		Funktionstyp:			RHD (kurz für Relative Humidity)
		Instanz-ID:				hier 1 (in XML nachschauen)
		Aktion:					STATUS
		P1:						Relative Luftfeuchtigkeit 0-100 Vorkommastellen
		P2:						Relative Luftfeuchtigkeit 0-100 Nachkommastellen

	Telegram Statusabfrage:  	
	
	\xFD 12345.RHD.1.gSTATUS \xFE
	
	Antwort:  					\xFD 12345.RHD.1.rSTATUS.P1 \xFE
	P1:							Relative Luftfeuchtigkeit 0-100 Vorkommastellen
	P2:							Relative Luftfeuchtigkeit 0-100 Nachkommastellen

	(*------------------------------------------------------------*)
	Helligkeitssensor (Sensor):
	(*------------------------------------------------------------*)
	Telegram Event:  	
	
	\xFD 12345.BRS.23.STATUS.P1.P2 \xFE
	
		Funktionstyp:			BRS (kurz für Brightness Sensor)
		Instanz-ID:				hier 23 (in XML nachschauen)
		Aktion:					STATUS
		P1:						Relative Helligkeit 0-255 Vorkommastellen
		P2:						Relative Helligkeit 0-255 Nachkommastellen
	
	Telegram Statusabfrage:  	
	
	\xFD 12345.BRS.23.gSTATUS \xFE
	
	Antwort:  					\xFD 12345.BRS.23.rSTATUS.P1 \xFE
	P1:							Relative Helligkeit 0-255 Vorkommastellen
	P2:							Relative Helligkeit 0-255 Nachkommastellen

(*======================================================================================================================================*)
(* Alle Telegramme im Überblick *)	

	<?xml version="1.0" encoding="utf-8"?>
	<Comm Title="Haus-Bus ID 1212" Comment="" Baudrate="57600" Databits="8" Parity="1" EndChar="510">
	<CommCmd Title="16-fach Relais 1212 - Rote Modul LED" Comment="" CmdOn="\xFD1212.OUT.210.ON.0\xFE" CmdOff="\xFD1212.OUT.210.OFF\xFE" Unit="" Analog="false" Text="false" Sensor="false" SourceValHigh="100" DestValHigh="100"/>
	<CommCmd Title="16-fach Relais 1212 - Relais 1" Comment="" CmdOn="\xFD1212.OUT.17.ON.0\xFE" CmdOff="\xFD1212.OUT.17.OFF\xFE" Unit="" Analog="false" Text="false" Sensor="false" SourceValHigh="100" DestValHigh="100"/>
	<CommCmd Title="16-fach Relais 1212 - Relais 2" Comment="" CmdOn="\xFD1212.OUT.18.ON.0\xFE" CmdOff="\xFD1212.OUT.18.OFF\xFE" Unit="" Analog="false" Text="false" Sensor="false" SourceValHigh="100" DestValHigh="100"/>
	<CommCmd Title="16-fach Relais 1212 - Relais 3" Comment="" CmdOn="\xFD1212.OUT.19.ON.0\xFE" CmdOff="\xFD1212.OUT.19.OFF\xFE" Unit="" Analog="false" Text="false" Sensor="false" SourceValHigh="100" DestValHigh="100"/>
	<CommCmd Title="16-fach Relais 1212 - Relais 4" Comment="" CmdOn="\xFD1212.OUT.20.ON.0\xFE" CmdOff="\xFD1212.OUT.20.OFF\xFE" Unit="" Analog="false" Text="false" Sensor="false" SourceValHigh="100" DestValHigh="100"/>
	<CommCmd Title="16-fach Relais 1212 - Relais 5" Comment="" CmdOn="\xFD1212.OUT.21.ON.0\xFE" CmdOff="\xFD1212.OUT.21.OFF\xFE" Unit="" Analog="false" Text="false" Sensor="false" SourceValHigh="100" DestValHigh="100"/>
	<CommCmd Title="16-fach Relais 1212 - Relais 6" Comment="" CmdOn="\xFD1212.OUT.22.ON.0\xFE" CmdOff="\xFD1212.OUT.22.OFF\xFE" Unit="" Analog="false" Text="false" Sensor="false" SourceValHigh="100" DestValHigh="100"/>
	<CommCmd Title="16-fach Relais 1212 - Relais 7" Comment="" CmdOn="\xFD1212.OUT.23.ON.0\xFE" CmdOff="\xFD1212.OUT.23.OFF\xFE" Unit="" Analog="false" Text="false" Sensor="false" SourceValHigh="100" DestValHigh="100"/>
	<CommCmd Title="16-fach Relais 1212 - Relais 8" Comment="" CmdOn="\xFD1212.OUT.24.ON.0\xFE" CmdOff="\xFD1212.OUT.24.OFF\xFE" Unit="" Analog="false" Text="false" Sensor="false" SourceValHigh="100" DestValHigh="100"/>
	<CommCmd Title="16-fach Relais 1212 - Relais 9" Comment="" CmdOn="\xFD1212.OUT.33.ON.0\xFE" CmdOff="\xFD1212.OUT.33.OFF\xFE" Unit="" Analog="false" Text="false" Sensor="false" SourceValHigh="100" DestValHigh="100"/>
	<CommCmd Title="16-fach Relais 1212 - Relais 10" Comment="" CmdOn="\xFD1212.OUT.34.ON.0\xFE" CmdOff="\xFD1212.OUT.34.OFF\xFE" Unit="" Analog="false" Text="false" Sensor="false" SourceValHigh="100" DestValHigh="100"/>
	<CommCmd Title="16-fach Relais 1212 - Relais 11" Comment="" CmdOn="\xFD1212.OUT.35.ON.0\xFE" CmdOff="\xFD1212.OUT.35.OFF\xFE" Unit="" Analog="false" Text="false" Sensor="false" SourceValHigh="100" DestValHigh="100"/>
	<CommCmd Title="16-fach Relais 1212 - Relais 12" Comment="" CmdOn="\xFD1212.OUT.36.ON.0\xFE" CmdOff="\xFD1212.OUT.36.OFF\xFE" Unit="" Analog="false" Text="false" Sensor="false" SourceValHigh="100" DestValHigh="100"/>
	<CommCmd Title="16-fach Relais 1212 - Relais 13" Comment="" CmdOn="\xFD1212.OUT.37.ON.0\xFE" CmdOff="\xFD1212.OUT.37.OFF\xFE" Unit="" Analog="false" Text="false" Sensor="false" SourceValHigh="100" DestValHigh="100"/>
	<CommCmd Title="16-fach Relais 1212 - Relais 14" Comment="" CmdOn="\xFD1212.OUT.38.ON.0\xFE" CmdOff="\xFD1212.OUT.38.OFF\xFE" Unit="" Analog="false" Text="false" Sensor="false" SourceValHigh="100" DestValHigh="100"/>
	<CommCmd Title="16-fach Relais 1212 - Relais 15" Comment="" CmdOn="\xFD1212.OUT.39.ON.0\xFE" CmdOff="\xFD1212.OUT.39.OFF\xFE" Unit="" Analog="false" Text="false" Sensor="false" SourceValHigh="100" DestValHigh="100"/>
	<CommCmd Title="16-fach Relais 1212 - Relais 16" Comment="" CmdOn="\xFD1212.OUT.40.ON.0\xFE" CmdOff="\xFD1212.OUT.40.OFF\xFE" Unit="" Analog="false" Text="false" Sensor="false" SourceValHigh="100" DestValHigh="100"/>
	<CommCmd Title="16-fach Relais 1212 - Eingang 1" Comment="" CmdOn="\xFD1212.BTN.97.STATUS.\v\xFE" CmdOff="" Unit="&lt;v.x&gt;" Analog="true" Text="false" Sensor="true" SourceValHigh="100" DestValHigh="100"/>
	<CommCmd Title="16-fach Relais 1212 - Eingang 2" Comment="" CmdOn="\xFD1212.BTN.98.STATUS.\v\xFE" CmdOff="" Unit="&lt;v.x&gt;" Analog="true" Text="false" Sensor="true" SourceValHigh="100" DestValHigh="100"/>
	<CommCmd Title="16-fach Relais 1212 - Eingang 3" Comment="" CmdOn="\xFD1212.BTN.99.STATUS.\v\xFE" CmdOff="" Unit="&lt;v.x&gt;" Analog="true" Text="false" Sensor="true" SourceValHigh="100" DestValHigh="100"/>
	<CommCmd Title="16-fach Relais 1212 - Eingang 4" Comment="" CmdOn="\xFD1212.BTN.100.STATUS.\v\xFE" CmdOff="" Unit="&lt;v.x&gt;" Analog="true" Text="false" Sensor="true" SourceValHigh="100" DestValHigh="100"/>
	<CommCmd Title="16-fach Relais 1212 - Eingang 5" Comment="" CmdOn="\xFD1212.BTN.101.STATUS.\v\xFE" CmdOff="" Unit="&lt;v.x&gt;" Analog="true" Text="false" Sensor="true" SourceValHigh="100" DestValHigh="100"/>
	<CommCmd Title="16-fach Relais 1212 - Eingang 6" Comment="" CmdOn="\xFD1212.BTN.102.STATUS.\v\xFE" CmdOff="" Unit="&lt;v.x&gt;" Analog="true" Text="false" Sensor="true" SourceValHigh="100" DestValHigh="100"/>
	<CommCmd Title="16-fach Relais 1212 - Eingang 7" Comment="" CmdOn="\xFD1212.BTN.103.STATUS.\v\xFE" CmdOff="" Unit="&lt;v.x&gt;" Analog="true" Text="false" Sensor="true" SourceValHigh="100" DestValHigh="100"/>
	<CommCmd Title="16-fach Relais 1212 - Eingang 8" Comment="" CmdOn="\xFD1212.BTN.104.STATUS.\v\xFE" CmdOff="" Unit="&lt;v.x&gt;" Analog="true" Text="false" Sensor="true" SourceValHigh="100" DestValHigh="100"/>
	</Comm>

*)
END_ACTION

END_FUNCTION_BLOCK

// ---- POUs/RS485_Hausbus_FB/RelaisModul/fb_StringConvRB16F.TcPOU
(*======================================================================================================================================*)
(*fb_StringConvRB16F:	Zusammensetzen des Strings für 16Fach Bus Relaismodul		*)
(*
Date          	| Version    	| created under        	| Author          	| Remark *)
(*====================================================================================================================================================*)
(*08/05/2025   	| 1.00      		| TC3		  		| N.Kersting       | first release *)
(*====================================================================================================================================================*)
FUNCTION_BLOCK fb_StringConvRB16F
VAR_INPUT
	I_bReset			:BOOL;							(* Reset Befehl auslösen *)
	I_bRedLEDOn			:BOOL;							(* Schaltet nur die Rote Modul LED ein*)
	I_bRedLEDOff		:BOOL;							(* Schaltet nur die Rote Modul LED aus*)
	I_diID				:DINT;							(* Device ID *)
	I_bOut    	 		:ARRAY[1..16] OF BOOL;     	  	(* gewünschter Relais zustand (TRUE = An %)*)
	
	I_iSection			:INT :=1;							(* Paarweise Schalten 1= 1&2 2= 3&4 usw. *)
	
	I_sStartZeichen		:BYTE := 16#FD;					(* Startzeichen Präfix *)
	I_sEndZeichen		:BYTE := 16#FE;					(* Endzeichen Suffix *)
END_VAR
VAR_OUTPUT
	Q_sConvString		:STRING(255);
END_VAR
VAR
	iStartOut			:INT := 1;
	iStartInstIDExt		:INT :=65;
	
END_VAR

IF NOT I_bReset
THEN
	IF I_bRedLEDOn
	THEN
		(* Rote Modul LED Ein*)
		iStartInstIDExt := 210;
		
		Q_sConvString:=	CONCAT(F_ToCHR(I_sStartZeichen),DINT_TO_STRING(I_diID));
		Q_sConvString:=	CONCAT(Q_sConvString,'.OUT.');
		Q_sConvString:=	CONCAT(Q_sConvString,INT_TO_STRING(iStartInstIDExt));
		Q_sConvString:=	CONCAT(Q_sConvString,'.ON');
		Q_sConvString:=	CONCAT(Q_sConvString,F_ToCHR(I_sEndZeichen));
	ELSIF
		I_bRedLEDOff
	THEN
		(* Rote Modul LED Aus*)
		iStartInstIDExt := 210;
		
		Q_sConvString:=	CONCAT(F_ToCHR(I_sStartZeichen),DINT_TO_STRING(I_diID));
		Q_sConvString:=	CONCAT(Q_sConvString,'.OUT.');
		Q_sConvString:=	CONCAT(Q_sConvString,INT_TO_STRING(iStartInstIDExt));
		Q_sConvString:=	CONCAT(Q_sConvString,'.OFF');
		Q_sConvString:=	CONCAT(Q_sConvString,F_ToCHR(I_sEndZeichen));
	ELSE
		CASE I_iSection OF
			
		0:	Q_sConvString:='';
		
		1:	(* 1 & 2 Schalten *)
			iStartInstIDExt := 17;
			iStartOut :=	1;
			
			Q_sConvString:=	CONCAT(F_ToCHR(I_sStartZeichen),DINT_TO_STRING(I_diID));
			Q_sConvString:=	CONCAT(Q_sConvString,'.OUT.');
			Q_sConvString:=	CONCAT(Q_sConvString,INT_TO_STRING(iStartInstIDExt));
			IF I_bOut[iStartOut]
			THEN
				Q_sConvString:=	CONCAT(Q_sConvString,'.ON');
			ELSE
				Q_sConvString:=	CONCAT(Q_sConvString,'.OFF');
			END_IF
			Q_sConvString:=	CONCAT(Q_sConvString,F_ToCHR(I_sEndZeichen));
			
			(* ##2 ##*)
			iStartInstIDExt := iStartInstIDExt +1;
			iStartOut:= iStartOut+1;
			
			Q_sConvString:=	CONCAT(Q_sConvString,F_ToCHR(I_sStartZeichen));
			Q_sConvString:=	CONCAT(Q_sConvString,DINT_TO_STRING(I_diID));
			Q_sConvString:=	CONCAT(Q_sConvString,'.OUT.');
			Q_sConvString:=	CONCAT(Q_sConvString,INT_TO_STRING(iStartInstIDExt));
			IF I_bOut[iStartOut]
			THEN
				Q_sConvString:=	CONCAT(Q_sConvString,'.ON');
			ELSE
				Q_sConvString:=	CONCAT(Q_sConvString,'.OFF');
			END_IF
			Q_sConvString:=	CONCAT(Q_sConvString,F_ToCHR(I_sEndZeichen));
		
			(* ##3 ##*)
			iStartInstIDExt := iStartInstIDExt +1;
			iStartOut:= iStartOut+1;
			
			Q_sConvString:=	CONCAT(Q_sConvString,F_ToCHR(I_sStartZeichen));
			Q_sConvString:=	CONCAT(Q_sConvString,DINT_TO_STRING(I_diID));
			Q_sConvString:=	CONCAT(Q_sConvString,'.OUT.');
			Q_sConvString:=	CONCAT(Q_sConvString,INT_TO_STRING(iStartInstIDExt));
			IF I_bOut[iStartOut]
			THEN
				Q_sConvString:=	CONCAT(Q_sConvString,'.ON');
			ELSE
				Q_sConvString:=	CONCAT(Q_sConvString,'.OFF');
			END_IF
			Q_sConvString:=	CONCAT(Q_sConvString,F_ToCHR(I_sEndZeichen));
			
			(* ##4 ##*)
			iStartInstIDExt := iStartInstIDExt +1;
			iStartOut:= iStartOut+1;
			
			Q_sConvString:=	CONCAT(Q_sConvString,F_ToCHR(I_sStartZeichen));
			Q_sConvString:=	CONCAT(Q_sConvString,DINT_TO_STRING(I_diID));
			Q_sConvString:=	CONCAT(Q_sConvString,'.OUT.');
			Q_sConvString:=	CONCAT(Q_sConvString,INT_TO_STRING(iStartInstIDExt));
			IF I_bOut[iStartOut]
			THEN
				Q_sConvString:=	CONCAT(Q_sConvString,'.ON');
			ELSE
				Q_sConvString:=	CONCAT(Q_sConvString,'.OFF');
			END_IF
			Q_sConvString:=	CONCAT(Q_sConvString,F_ToCHR(I_sEndZeichen));
		
			(* ##5 ##*)
			iStartInstIDExt := iStartInstIDExt +1;
			iStartOut:= iStartOut+1;
			
			Q_sConvString:=	CONCAT(Q_sConvString,F_ToCHR(I_sStartZeichen));
			Q_sConvString:=	CONCAT(Q_sConvString,DINT_TO_STRING(I_diID));
			Q_sConvString:=	CONCAT(Q_sConvString,'.OUT.');
			Q_sConvString:=	CONCAT(Q_sConvString,INT_TO_STRING(iStartInstIDExt));
			IF I_bOut[iStartOut]
			THEN
				Q_sConvString:=	CONCAT(Q_sConvString,'.ON');
			ELSE
				Q_sConvString:=	CONCAT(Q_sConvString,'.OFF');
			END_IF
			Q_sConvString:=	CONCAT(Q_sConvString,F_ToCHR(I_sEndZeichen));
			
			(* ##6 ##*)
			iStartInstIDExt := iStartInstIDExt +1;
			iStartOut:= iStartOut+1;
			
			Q_sConvString:=	CONCAT(Q_sConvString,F_ToCHR(I_sStartZeichen));
			Q_sConvString:=	CONCAT(Q_sConvString,DINT_TO_STRING(I_diID));
			Q_sConvString:=	CONCAT(Q_sConvString,'.OUT.');
			Q_sConvString:=	CONCAT(Q_sConvString,INT_TO_STRING(iStartInstIDExt));
			IF I_bOut[iStartOut]
			THEN
				Q_sConvString:=	CONCAT(Q_sConvString,'.ON');
			ELSE
				Q_sConvString:=	CONCAT(Q_sConvString,'.OFF');
			END_IF
			Q_sConvString:=	CONCAT(Q_sConvString,F_ToCHR(I_sEndZeichen));
		
			(* ##7 ##*)
			iStartInstIDExt := iStartInstIDExt +1;
			iStartOut:= iStartOut+1;
			
			Q_sConvString:=	CONCAT(Q_sConvString,F_ToCHR(I_sStartZeichen));
			Q_sConvString:=	CONCAT(Q_sConvString,DINT_TO_STRING(I_diID));
			Q_sConvString:=	CONCAT(Q_sConvString,'.OUT.');
			Q_sConvString:=	CONCAT(Q_sConvString,INT_TO_STRING(iStartInstIDExt));
			IF I_bOut[iStartOut]
			THEN
				Q_sConvString:=	CONCAT(Q_sConvString,'.ON');
			ELSE
				Q_sConvString:=	CONCAT(Q_sConvString,'.OFF');
			END_IF
			Q_sConvString:=	CONCAT(Q_sConvString,F_ToCHR(I_sEndZeichen));
			
			(* ##8 ##*)
			iStartInstIDExt := iStartInstIDExt +1;
			iStartOut:= iStartOut+1;
			
			Q_sConvString:=	CONCAT(Q_sConvString,F_ToCHR(I_sStartZeichen));
			Q_sConvString:=	CONCAT(Q_sConvString,DINT_TO_STRING(I_diID));
			Q_sConvString:=	CONCAT(Q_sConvString,'.OUT.');
			Q_sConvString:=	CONCAT(Q_sConvString,INT_TO_STRING(iStartInstIDExt));
			IF I_bOut[iStartOut]
			THEN
				Q_sConvString:=	CONCAT(Q_sConvString,'.ON');
			ELSE
				Q_sConvString:=	CONCAT(Q_sConvString,'.OFF');
			END_IF
			Q_sConvString:=	CONCAT(Q_sConvString,F_ToCHR(I_sEndZeichen));
		
		2:	(* 9 & 10 Schalten *)
			iStartInstIDExt := 33;
			iStartOut :=	9;
			
			Q_sConvString:=	CONCAT(F_ToCHR(I_sStartZeichen),DINT_TO_STRING(I_diID));
			Q_sConvString:=	CONCAT(Q_sConvString,'.OUT.');
			Q_sConvString:=	CONCAT(Q_sConvString,INT_TO_STRING(iStartInstIDExt));
			IF I_bOut[iStartOut]
			THEN
				Q_sConvString:=	CONCAT(Q_sConvString,'.ON');
			ELSE
				Q_sConvString:=	CONCAT(Q_sConvString,'.OFF');
			END_IF
			Q_sConvString:=	CONCAT(Q_sConvString,F_ToCHR(I_sEndZeichen));
			
			(* ##10 ##*)
			iStartInstIDExt := iStartInstIDExt +1;
			iStartOut:= iStartOut+1;
			
			Q_sConvString:=	CONCAT(Q_sConvString,F_ToCHR(I_sStartZeichen));
			Q_sConvString:=	CONCAT(Q_sConvString,DINT_TO_STRING(I_diID));
			Q_sConvString:=	CONCAT(Q_sConvString,'.OUT.');
			Q_sConvString:=	CONCAT(Q_sConvString,INT_TO_STRING(iStartInstIDExt));
			IF I_bOut[iStartOut]
			THEN
				Q_sConvString:=	CONCAT(Q_sConvString,'.ON');
			ELSE
				Q_sConvString:=	CONCAT(Q_sConvString,'.OFF');
			END_IF
			Q_sConvString:=	CONCAT(Q_sConvString,F_ToCHR(I_sEndZeichen));
		
			(* ##11 ##*)
			iStartInstIDExt := iStartInstIDExt +1;
			iStartOut:= iStartOut+1;
			
			Q_sConvString:=	CONCAT(Q_sConvString,F_ToCHR(I_sStartZeichen));
			Q_sConvString:=	CONCAT(Q_sConvString,DINT_TO_STRING(I_diID));
			Q_sConvString:=	CONCAT(Q_sConvString,'.OUT.');
			Q_sConvString:=	CONCAT(Q_sConvString,INT_TO_STRING(iStartInstIDExt));
			IF I_bOut[iStartOut]
			THEN
				Q_sConvString:=	CONCAT(Q_sConvString,'.ON');
			ELSE
				Q_sConvString:=	CONCAT(Q_sConvString,'.OFF');
			END_IF
			Q_sConvString:=	CONCAT(Q_sConvString,F_ToCHR(I_sEndZeichen));
			
			(* ##12 ##*)
			iStartInstIDExt := iStartInstIDExt +1;
			iStartOut:= iStartOut+1;
			
			Q_sConvString:=	CONCAT(Q_sConvString,F_ToCHR(I_sStartZeichen));
			Q_sConvString:=	CONCAT(Q_sConvString,DINT_TO_STRING(I_diID));
			Q_sConvString:=	CONCAT(Q_sConvString,'.OUT.');
			Q_sConvString:=	CONCAT(Q_sConvString,INT_TO_STRING(iStartInstIDExt));
			IF I_bOut[iStartOut]
			THEN
				Q_sConvString:=	CONCAT(Q_sConvString,'.ON');
			ELSE
				Q_sConvString:=	CONCAT(Q_sConvString,'.OFF');
			END_IF
			Q_sConvString:=	CONCAT(Q_sConvString,F_ToCHR(I_sEndZeichen));
		
			(* ##13 ##*)
			iStartInstIDExt := iStartInstIDExt +1;
			iStartOut:= iStartOut+1;
			
			Q_sConvString:=	CONCAT(Q_sConvString,F_ToCHR(I_sStartZeichen));
			Q_sConvString:=	CONCAT(Q_sConvString,DINT_TO_STRING(I_diID));
			Q_sConvString:=	CONCAT(Q_sConvString,'.OUT.');
			Q_sConvString:=	CONCAT(Q_sConvString,INT_TO_STRING(iStartInstIDExt));
			IF I_bOut[iStartOut]
			THEN
				Q_sConvString:=	CONCAT(Q_sConvString,'.ON');
			ELSE
				Q_sConvString:=	CONCAT(Q_sConvString,'.OFF');
			END_IF
			Q_sConvString:=	CONCAT(Q_sConvString,F_ToCHR(I_sEndZeichen));
			
			(* ##14 ##*)
			iStartInstIDExt := iStartInstIDExt +1;
			iStartOut:= iStartOut+1;
			
			Q_sConvString:=	CONCAT(Q_sConvString,F_ToCHR(I_sStartZeichen));
			Q_sConvString:=	CONCAT(Q_sConvString,DINT_TO_STRING(I_diID));
			Q_sConvString:=	CONCAT(Q_sConvString,'.OUT.');
			Q_sConvString:=	CONCAT(Q_sConvString,INT_TO_STRING(iStartInstIDExt));
			IF I_bOut[iStartOut]
			THEN
				Q_sConvString:=	CONCAT(Q_sConvString,'.ON');
			ELSE
				Q_sConvString:=	CONCAT(Q_sConvString,'.OFF');
			END_IF
			Q_sConvString:=	CONCAT(Q_sConvString,F_ToCHR(I_sEndZeichen));
		
			(* ##15 ##*)
			iStartInstIDExt := iStartInstIDExt +1;
			iStartOut:= iStartOut+1;
			
			Q_sConvString:=	CONCAT(Q_sConvString,F_ToCHR(I_sStartZeichen));
			Q_sConvString:=	CONCAT(Q_sConvString,DINT_TO_STRING(I_diID));
			Q_sConvString:=	CONCAT(Q_sConvString,'.OUT.');
			Q_sConvString:=	CONCAT(Q_sConvString,INT_TO_STRING(iStartInstIDExt));
			IF I_bOut[iStartOut]
			THEN
				Q_sConvString:=	CONCAT(Q_sConvString,'.ON');
			ELSE
				Q_sConvString:=	CONCAT(Q_sConvString,'.OFF');
			END_IF
			Q_sConvString:=	CONCAT(Q_sConvString,F_ToCHR(I_sEndZeichen));
			
			(* ##16 ##*)
			iStartInstIDExt := iStartInstIDExt +1;
			iStartOut:= iStartOut+1;
			
			Q_sConvString:=	CONCAT(Q_sConvString,F_ToCHR(I_sStartZeichen));
			Q_sConvString:=	CONCAT(Q_sConvString,DINT_TO_STRING(I_diID));
			Q_sConvString:=	CONCAT(Q_sConvString,'.OUT.');
			Q_sConvString:=	CONCAT(Q_sConvString,INT_TO_STRING(iStartInstIDExt));
			IF I_bOut[iStartOut]
			THEN
				Q_sConvString:=	CONCAT(Q_sConvString,'.ON');
			ELSE
				Q_sConvString:=	CONCAT(Q_sConvString,'.OFF');
			END_IF
			Q_sConvString:=	CONCAT(Q_sConvString,F_ToCHR(I_sEndZeichen));
		END_CASE
	END_IF
	
ELSE
	(* Reset *)
	Q_sConvString:=	CONCAT(F_ToCHR(I_sStartZeichen),DINT_TO_STRING(I_diID));
	Q_sConvString:=	CONCAT(Q_sConvString,'.SYS.');
	Q_sConvString:=	CONCAT(Q_sConvString,INT_TO_STRING(1));
	Q_sConvString:=	CONCAT(Q_sConvString,'.RESET');
	Q_sConvString:=	CONCAT(Q_sConvString,F_ToCHR(I_sEndZeichen));
END_IF

END_FUNCTION_BLOCK

// ---- POUs/RS485_Hausbus_FB/RS485 COM/RS485_Master/fb_RS485Startup.TcPOU
(*======================================================================================================================================*)
(*fb_RS485Startup:	Einfacher Baustein um die Hardware für die RS485 Haus-Bus vorzubereiten*)
(*
Date          	| Version    	| created under        	| Author          	| Remark *)
(*====================================================================================================================================================*)
(*13/05/2025   	| 1.00      		| TC3		  		| N.Kersting       | first release *)
(*====================================================================================================================================================*)
FUNCTION_BLOCK fb_RS485Startup
VAR_INPUT
	I_bExecute						:BOOL;
	I_bBusOK						:BOOL;
	I_tStartupVerz					:TIME := T#2S;	(* Startup verzögert ausführen *)
END_VAR
VAR_IN_OUT
	IQ_InData	 					:KL6inData22B;
    IQ_OutData						:KL6outData22B;
END_VAR
VAR_OUTPUT
	Q_sState						:STRING;
	Q_bStartupDone					:BOOL;
	Q_bError						:BOOL;
	Q_stStates						:ST_RS485Startup_State;
END_VAR
VAR
	udBaudrate						:UDINT := 57600;
	byDataBits						:BYTE := 8;
	byStopBits						:BYTE := 1;
	
	tonStartupVerz					:ton;
	fbSerialComReset				:ComReset;
	fComBufferReset					:ClearComBuffer;
	fbSerialConfig 					:KL6Configuration;  // Terminal-Konfiguration (Baud, Parität etc.)
	iStepStartup					:INT;
END_VAR

tonStartupVerz(
	PT :=	I_tStartupVerz);
	
CASE iStepStartup OF 
(*=========================================================================*)
0:	IF NOT Q_bError
		AND I_bBusOK
	THEN
		Q_sState := 'INIT';
	ELSIF
		NOT I_bBusOK
	THEN
		Q_bError := TRUE;
		Q_sState := 'Busverbindung nicht Ok';
	END_IF
	
	tonStartupVerz.IN := FALSE;
	
	fbSerialComReset(
		Execute:= 		FALSE);
		
	fbSerialConfig(
		Execute:= 		FALSE);
		
	IF I_bExecute
		AND I_bBusOK
	THEN
		Q_bStartupDone := FALSE;
		iStepStartup := iStepStartup+1;
	END_IF

(*=========================================================================*)
1:	Q_sState := 'Warten auf Verzögerung';
	tonStartupVerz.IN := TRUE; 
	
	IF tonStartupVerz.Q
	THEN
		iStepStartup := iStepStartup+1;
	END_IF
	
(*=========================================================================*)
2:	Q_sState := 'Serielle Klemme Konfigurieren mit Haus-Bus Vorgaben';	
	
	fbSerialConfig(
		Execute:= 		TRUE, 
		Mode:= 			ComSerialLineMode_t.SERIALLINEMODE_KL6_22B_STANDARD,		 
		Baudrate:= 		udBaudrate, 
		NoDatabits:= 	byDataBits, 
		Parity:= 		ComParity_t.PARITY_EVEN,	 
		Stopbits:= 		byStopBits, 
		Handshake:= 	RS485_HALFDUPLEX, 
		ContinousMode:= , 
		pComIn := 		ADR(IQ_InData), 
		pComOut := 		ADR(IQ_OutData), 
		SizeComIn := 	SIZEOF(IQ_InData),
		Done=> , 
		Busy=> , 
		Error=> , 
		ErrorId=> );
	
	IF fbSerialConfig.Done
	THEN
		fbSerialConfig(
			Execute:= 		FALSE); 
			
		iStepStartup := 3;
	ELSIF
		fbSerialConfig.Error
	THEN
		Q_sState := 'Error fbSerialConfig ID: ';
		Q_sState := CONCAT(Q_sState,INT_TO_STRING(fbSerialConfig.ErrorID));
		iStepStartup := -2;	//Error
	END_IF

(*=========================================================================*)
3:	Q_sState := 'Serielle Klemme Reset Auführen';	
		
	fbSerialComReset(
		Execute:= 		TRUE, 
		pComIn := 		ADR(IQ_InData), 
		pComOut := 		ADR(IQ_OutData), 
		SizeComIn := 	SIZEOF(IQ_InData),
		Done=> , 
		Busy=> , 
		Error=> , 
		ErrorID=> );	
		
	IF fbSerialComReset.Done
	THEN
		iStepStartup := 999;
	ELSIF
		fbSerialComReset.Error
	THEN
		Q_sState := 'Error fbSerialComReset ID: ';
		Q_sState := CONCAT(Q_sState,INT_TO_STRING(fbSerialComReset.ErrorID));
		iStepStartup := -3;	//Error
	END_IF
	
(*=========================================================================*)
999:Q_sState := 'Startup Ausgeführt!';	
	Q_bStartupDone := TRUE;
	Q_bError := FALSE;
	
	IF NOT I_bBusOK
	THEN
		Q_bStartupDone := FALSE;
		iStepStartup := 0;
	END_IF

ELSE
	(* ERROR *)
	Q_bError := TRUE;
	iStepStartup := 0;
END_CASE

(* StatusStruktur für Visu *)
Q_stStates.bBusOk				:=	I_bBusOK;
Q_stStates.bStartupDone			:=	Q_bStartupDone;
Q_stStates.bStartupError		:=	Q_bError;
Q_stStates.sStartupState		:=	Q_sState;

END_FUNCTION_BLOCK

// ---- POUs/RS485_Hausbus_FB/RS485 COM/RS485_Master/fb_RS485FiFoMaster.TcPOU
(*======================================================================================================================================*)
(*fb_RS485FiFoMaster:	Einfaches Senden eines Telegrams über RS485*)
(*
Date          	| Version    	| created under        	| Author          	| Remark *)
(*====================================================================================================================================================*)
(*10/05/2025   	| 1.00      		| TC3		  		| N.Kersting       | first release *)
(*10/05/2025   	| 1.01      		| TC3		  		| N.Kersting       | Nun wird der Empfang auch mit Implementiert  *)
(*13/05/2025   	| 1.02      		| TC3		  		| N.Kersting       | Busbelastungstest Implementiert - Sendet Durchgehend Strings *)
(*14/05/2025   	| 1.03      		| TC3		  		| N.Kersting       | Busauslastung direkt Implementiert *)
(*====================================================================================================================================================*)
FUNCTION_BLOCK fb_RS485FiFoMaster
VAR_INPUT
	I_sSendCmdFiFo				:ARRAY[1..cMaxRS485CMDFiFo] OF STRING(255);
	I_bExecute					:BOOL := TRUE;
	I_bBusBelastungstest		:BOOL;
	I_bReset					:BOOL;
	I_pTxBuffer					:POINTER TO ComBuffer;  (*Zeiger auf TX-Buffer*)
	I_pRxBuffer   				:POINTER TO ComBuffer;  (*Zeiger auf RX-Buffer*)
END_VAR
VAR_OUTPUT
	Q_sReceiveString			:STRING(255);		
	Q_lrBusAuslastung			:LREAL;
	Q_bBusy						:BOOL;
	Q_bDone						:BOOL;
	Q_bError					:BOOL;
	Q_sState					:STRING;
	Q_stStates					:ST_FiFoMaster_State;
END_VAR
VAR
	bFirstCycle					:BOOL := TRUE;
	tVerzReceive				:TIME := T#30MS;			(* Zeit, die zum Empfangen bleibt *)
	
	tonSend						:ton;
	fbSend     					:SendString255;
	fbReceive   				:ReceiveString255;
	sStartZeichen				:BYTE := 16#FD;				(* Startzeichen Präfix *)
	sEndZeichen					:BYTE := 16#FE;				(* Endzeichen Suffix *)
	sReceivedMEMString			:STRING(255);
	sReceivedString				:STRING(255);
	iStep						:INT;
	iStepReceive				:INT;
	iMaxBufferBlocking			:INT := 0;
	bBusyMem					:BOOL;
	sStep						:STRING;
	sString						:STRING(255);
	sStringSend					:STRING(255);
	tonVerzReceive				:ton;	
	tonTimeout					:ton;
	bStringSend					:BOOL := FALSE;
	icntError					:INT;
	
	iFiFoRow					:INT := 1;
	icntFiFo					:INT;
	i,h							:INT;
	iStepFiFo					:INT;
	
	bBusBelastungstest			:BOOL := FALSE;
	bBusAuslastung				:BOOL := TRUE;
	fbBusAuslastung				:fb_FilterArray;
END_VAR

(*============================================================================================*)
tonTimeout(
	PT:=T#1S);
	
tonVerzReceive(
	pt := tVerzReceive);

(* Busbelastungstest *)	
bBusBelastungstest := I_bBusBelastungstest;

sReceivedMEMString:='';
(*============================================================================================*)	
icntFiFo := 0;
FOR i := 1 TO cMaxRS485CMDFiFo BY 1 DO 
	IF (I_sSendCmdFiFo[i]<> '')
	THEN
		icntFiFo := icntFiFo +1;
	END_IF
END_FOR

(*============================================================================================*)
CASE iStepFiFo OF
-1:	sStep := 'FiFo INIT';
	bFirstCycle := FALSE;
	Q_bBusy := FALSE;
	iFiFoRow := 1;
	
	FOR h := 1 TO cMaxRS485CMDFiFo BY 1 DO
		GVL_RS485FiFoSend.bSendDoneFiFo[h] :=TRUE;
	END_FOR
	
	iStepFiFo := 0;

(*============================================================================================*)
0:	sStep := 'Warten, dass FiFo gefüllt wird';
	iFiFoRow := 1;
	bStringSend := FALSE;
	Q_bBusy := FALSE;
	tonVerzReceive.IN := (I_pTxBuffer^.Count<= INT_TO_UINT(iMaxBufferBlocking));
	
	IF (icntFiFo > 0
		OR  bBusBelastungstest)
		AND NOT bFirstCycle
		AND NOT fbReceive.StringReceived
		AND tonVerzReceive.Q
	THEN
		Q_bBusy := TRUE;
		iStepFiFo := 1;
	ELSIF
		bFirstCycle
	THEN
		iStepFiFo := -1;
	END_IF
	
(*============================================================================================*)	
1:	sStep := 'Prüfen ob STRING in FiFo Zeile gefüllt*';
	sStringSend :=	I_sSendCmdFiFo[iFiFoRow]; 
	
	(* Prüfen ob in der ausgewählten Zeile etwas steht *)
	IF I_sSendCmdFiFo[iFiFoRow] = ''
	THEN
		IF iFiFoRow < cMaxRS485CMDFiFo
		THEN
			iFiFoRow := iFiFoRow+1; (* Nächste Zeile, bis etwas drin Steht *)
		ELSE
			IF bBusBelastungstest
			THEN
				sStringSend :=	CONCAT(F_ToCHR(sStartZeichen),'ServiceTOOL-BUSBELASTUNGSTEST-BURSTFIREMODE');
				sStringSend :=	CONCAT(sStringSend,F_ToCHR(sEndZeichen));
				(* Senden *)
				
				IF NOT I_pTxBuffer^.blocked
					AND (I_pTxBuffer^.Error=0)
					AND NOT fbReceive.StringReceived
				THEN
					sStep := 'Prüfe ob Senden noch aktiv ist';
					bStringSend := TRUE;
					sString :=	sStringSend;
					Q_bDone := FALSE;
					Q_bError := FALSE;
					iStepFiFo := iStepFiFo+1;
				END_IF
			ELSE
				iStepFiFo := 0;	(* Alle Zeilen Abgearbeitet *)
			END_IF
			
		END_IF
	ELSE
		(* Senden *)
		GVL_RS485FiFoSend.bSendDoneFiFo[iFiFoRow] :=FALSE;
		
		IF NOT I_pTxBuffer^.blocked
			AND (I_pTxBuffer^.Error=0)
			AND NOT fbReceive.StringReceived
		THEN
			sStep := 'Prüfe ob Senden noch aktiv ist';
			bStringSend := TRUE;
			sString :=	sStringSend;
			Q_bDone := FALSE;
			Q_bError := FALSE;
			iStepFiFo := iStepFiFo+1;
		END_IF
	END_IF
	
(*============================================================================================*)		
2:	sStep := 'Starte Senden';
	Q_bBusy := TRUE;
	tonTimeout.IN := fbSend.Busy;
	
	IF NOT fbSend.Busy
		AND NOT fbReceive.StringReceived
	THEN
		tonSend.IN := FALSE;
		bStringSend := FALSE;
		iStepFiFo := iStepFiFo+1;
	ELSIF
		(fbSend.Error >0)
		AND NOT (fbSend.Error = 2)
	THEN
		sStep := CONCAT('ERROR-',sStep);
		sStep := CONCAT(sStep,'- ');
		sStep := CONCAT(sStep,INT_TO_STRING(fbSend.Error));
		iStepFiFo := -2;
	ELSIF
		tonTimeout.Q
	THEN
		sStep := CONCAT('ERROR- Timeout',sStep);
		iStepFiFo := -2;
	END_IF

3:	(* Senden*)		
	GVL_RS485FiFoSend.bSendDoneFiFo[iFiFoRow] :=TRUE;
	
	IF iFiFoRow < iFiFoRow
	THEN
		iFiFoRow := iFiFoRow+1;
		iStepFiFo := 1;
	ELSE
		Q_bDone := TRUE;
		iStepFiFo := 0;
	END_IF

ELSE
(*============================================================================================*)
	Q_bError := TRUE;
	Q_bBusy := FALSE;
	bBusyMem := FALSE;
	tonTimeout.IN := FALSE;
	
	IF I_bReset
	THEN
		iStepFiFo := 0;
	END_IF
END_CASE

IF bStringSend
THEN
	fbSend(
		SendString:= 	sString,
		TXbuffer:= 		I_pTxBuffer^);
ELSE
	(* Empfangen *)
	ac00_Receive();
END_IF

(* Empfangsmerker 0 Setzen am ende Eines Zyklus *)
Q_sReceiveString := sReceivedMEMString;

(* Busauslastung tracken*)
ac99_Diagnose();

Q_sState :=	sStep;

(* StatusStruktur für Visu *)
Q_stStates.bBusy				:=	Q_bBusy;
Q_stStates.bDone				:=	Q_bDone;
Q_stStates.bError				:=	Q_bError;
Q_stStates.iFiFoCount			:=	icntFiFo;
Q_stStates.iFiFoRow				:=	iFiFoRow;
Q_stStates.lrBusAuslastung		:=	Q_lrBusAuslastung;
Q_stStates.sReceiveString 		:=	Q_sReceiveString;
Q_stStates.sSendString 			:=	sString;
Q_stStates.sState 				:=	Q_sState;

ACTION ac00_Receive:
(* Empfangen *)
CASE iStepReceive OF		
0:	fbReceive(
		Prefix := 			F_ToCHR(sStartZeichen),
		Suffix := 			F_ToCHR(sEndZeichen),
		Timeout:= , 
		Reset:= , 
		StringReceived=> , 
		Busy=> , 
		Error=> , 
		RxTimeout=> , 
		ReceivedString:= 	sReceivedString, 
		RXbuffer:= 			I_pRxBuffer^);
		
	IF fbReceive.StringReceived
	THEN
		iStepReceive := 1;
		sReceivedMEMString := sReceivedString;
	END_IF
	
1:	sReceivedString := '';
	iStepReceive := 0;
	
END_CASE
END_ACTION

ACTION ac99_Diagnose:
(* Busauslastung Prüfen *)
fbBusAuslastung(
	I_bExcecute:= 	bBusAuslastung, 
	I_nWert:= 		UINT_TO_LREAL(I_pTxBuffer^.Count), 
	I_nFilterWert:= 50, 
	Q_nFilter=> 	Q_lrBusAuslastung);
END_ACTION

END_FUNCTION_BLOCK

// ---- POUs/RS485_Hausbus_FB/RS485 COM/FB/fb_FilterArray.TcPOU
(*======================================================================================================================================*)
(* Dieser Baustein Filtert eine Lreal Variable durch bildung eines Mittelwerts
(*======================================================================================================================================*)						

Date          		| Version    		| created under        		| Author          		| Remark *)
(*======================================================================================================================================*)
(*´10/07/2024   	| 1.00      			| TC2			  		| N.Kersting       	| first release *)
(*´15/07/2024   	| 1.01      			| TC2			  		| N.Kersting       	| Filterung nun Variabel einstellbar *)
(*======================================================================================================================================*)
FUNCTION_BLOCK fb_FilterArray
VAR_INPUT
	I_bExcecute	:BOOL;
	I_nWert		:LREAL;
	I_nFilterWert	:INT	:= 10;
END_VAR
VAR_OUTPUT
	Q_nFilter		:LREAL;
END_VAR
VAR
	i	:INT;
	nWertArray	:ARRAY [0..50] OF LREAL;
END_VAR

IF I_bExcecute THEN
   (* // Verschieben der Werte im Array*)
    FOR i := I_nFilterWert - 1 TO 1 BY -1 DO
        nWertArray[i] := nWertArray[i - 1];
    END_FOR

   (* // Neuen Wert einfügen	*)
    nWertArray[0] := I_nWert;

  (*  // Berechnung des gefilterten Wertes*)
    Q_nFilter := 0;
    FOR i := 0 TO I_nFilterWert - 1 DO
        Q_nFilter := Q_nFilter + nWertArray[i];
    END_FOR
    Q_nFilter := Q_nFilter / I_nFilterWert;

ELSE
  (*  // Initialisieren des Arrays*)
    FOR i := 0 TO 10 DO
        nWertArray[i] := 0;
    END_FOR
    Q_nFilter := 0;
END_IF

// ---- GlobalTextList.TcGTLO
TEXTLIST GlobalTextList
  573 = '%s'
  382 = 'BG LEDs: %s'
  258 = 'BTN1'
  576 = 'BTN1 %s'
  715 = 'BTN1Ext'
  297 = 'BTN2 '
  965 = 'BTN2 %s '
  554 = 'BTN2Ext'
  479 = 'BTN3'
  188 = 'BTN3 %s'
  737 = 'BTN3Ext'
  989 = 'BTN4'
  390 = 'BTN4 %s'
  345 = 'BTN4Ext'
  308 = 'BTN5'
  533 = 'BTN5 %s'
  511 = 'BTN5Ext'
  943 = 'BTN6'
  202 = 'BTN6 %s'
  907 = 'BTN6Ext'
  595 = 'BTN7'
  941 = 'BTN8'
  450 = 'Bus'
  874 = 'Bus Ok'
  355 = 'Busbelastungstest'
  902 = 'Busy'
  187 = 'COM'
  634 = 'Count %s '
  323 = 'Done'
  235 = 'Error'
  325 = "Externe E/A's"
  790 = 'FiFo Master'
  246 = 'Humi: %s p'
  180 = "Interne E/A's"
  925 = 'Interne Eingänge '
  921 = 'Lum: %s p'
  356 = 'R1'
  892 = 'R10'
  223 = 'R11'
  245 = 'R12'
  593 = 'R13'
  117 = 'R14'
  996 = 'R15'
  327 = 'R16'
  233 = 'R2'
  713 = 'R3'
  132 = 'R4'
  769 = 'R5'
  317 = 'R6'
  716 = 'R7'
  350 = 'R8'
  333 = 'R9'
  663 = 'Relais'
  267 = 'Relais '
  292 = 'Reset'
  342 = 'Row %s '
  289 = 'RX: %s'
  172 = 'Startup\nDone'
  38 = 'Startup\nError'
  25 = 'Startup :%s '
  789 = 'State :%s '
  93 = 'Taster'
  696 = 'Temp: %s °C'
  18 = 'TX: %s'
  58 = 'Visu Service Mode'
END_TEXTLIST

// ---- VISUs/HausBus_RS485/BusRelais16F_Frame.TcVIS
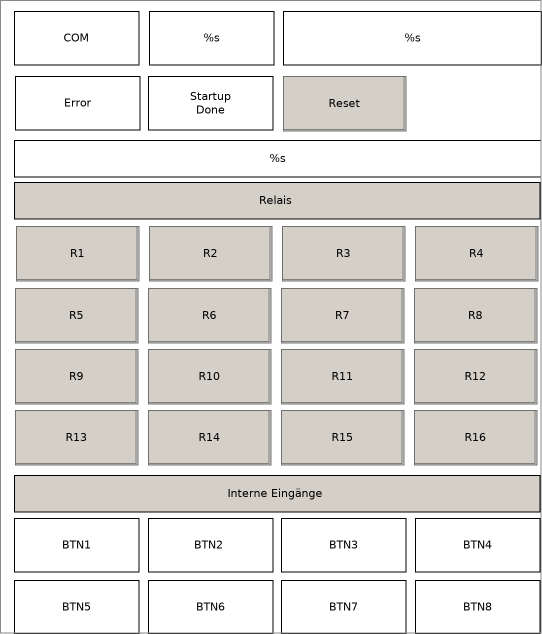
VISUALIZATION BusRelais16F_Frame  // 542x634
VAR_IN_OUT
	ST_BusRelais16F_Input		:ST_BusRelais16F_Input;
	ST_BusRelais16F_Output		:ST_BusRelais16F_Output;
	ST_BusRelais16F_Cnt			:ST_BusRelais16F_Cnt;
END_VAR
    Rectangle (14,11 125x54), "COM", colour toggle: ST_BusRelais16F_Output.bCOM
    Rectangle (14,518 125x54), "BTN1", colour toggle: ST_BusRelais16F_Output.bInputs[1]
    Rectangle (149,11 125x54), "%s", text variable: ST_BusRelais16F_Input.diID
    Rectangle (283,11 259x54), "%s", text variable: ST_BusRelais16F_Input.sName
    Rectangle (148,518 125x54), "BTN2", colour toggle: ST_BusRelais16F_Output.bInputs[2]
    Rectangle (281,518 125x54), "BTN3", colour toggle: ST_BusRelais16F_Output.bInputs[3]
    Rectangle (415,518 125x54), "BTN4", colour toggle: ST_BusRelais16F_Output.bInputs[4]
    Rectangle (14,580 125x54), "BTN5", colour toggle: ST_BusRelais16F_Output.bInputs[5]
    Rectangle (148,580 125x54), "BTN6", colour toggle: ST_BusRelais16F_Output.bInputs[6]
    Button (283,76 123x55), "Reset"
        tap ST_BusRelais16F_Input.bReset
    Rectangle (15,76 125x54), "Error", colour toggle: ST_BusRelais16F_Output.bError
    Rectangle (14,140 527x37), "%s", text variable: ST_BusRelais16F_Output.sState
    Rectangle (148,76 125x54), "Startup Done", colour toggle: ST_BusRelais16F_Output.bStartupDone
    Rectangle (14,475 526x37), "Interne Eingänge"
    Rectangle (281,580 125x54), "BTN7", colour toggle: ST_BusRelais16F_Output.bInputs[7]
    Rectangle (415,580 125x54), "BTN8", colour toggle: ST_BusRelais16F_Output.bInputs[8]
    Button (16,226 123x55), "R1"
        toggle ST_BusRelais16F_Input.bOut[1]
    Rectangle (14,182 526x37), "Relais"
    Button (149,226 123x55), "R2"
        toggle ST_BusRelais16F_Input.bOut[2]
    Button (282,226 123x55), "R3"
        toggle ST_BusRelais16F_Input.bOut[3]
    Button (415,226 123x55), "R4"
        toggle ST_BusRelais16F_Input.bOut[4]
    Button (15,288 123x55), "R5"
        toggle ST_BusRelais16F_Input.bOut[5]
    Button (148,288 123x55), "R6"
        toggle ST_BusRelais16F_Input.bOut[6]
    Button (281,288 123x55), "R7"
        toggle ST_BusRelais16F_Input.bOut[7]
    Button (414,288 123x55), "R8"
        toggle ST_BusRelais16F_Input.bOut[8]
    Button (15,349 123x55), "R9"
        toggle ST_BusRelais16F_Input.bOut[9]
    Button (148,349 123x55), "R10"
        toggle ST_BusRelais16F_Input.bOut[10]
    Button (281,349 123x55), "R11"
        toggle ST_BusRelais16F_Input.bOut[11]
    Button (414,349 123x55), "R12"
        toggle ST_BusRelais16F_Input.bOut[12]
    Button (15,410 123x55), "R13"
        toggle ST_BusRelais16F_Input.bOut[13]
    Button (148,410 123x55), "R14"
        toggle ST_BusRelais16F_Input.bOut[14]
    Button (281,410 123x55), "R15"
        toggle ST_BusRelais16F_Input.bOut[15]
    Button (414,410 123x55), "R16"
        toggle ST_BusRelais16F_Input.bOut[16]
END_VISUALIZATION

// ---- VISUs/HausBus_RS485/BusRS485Master_Frame.TcVIS
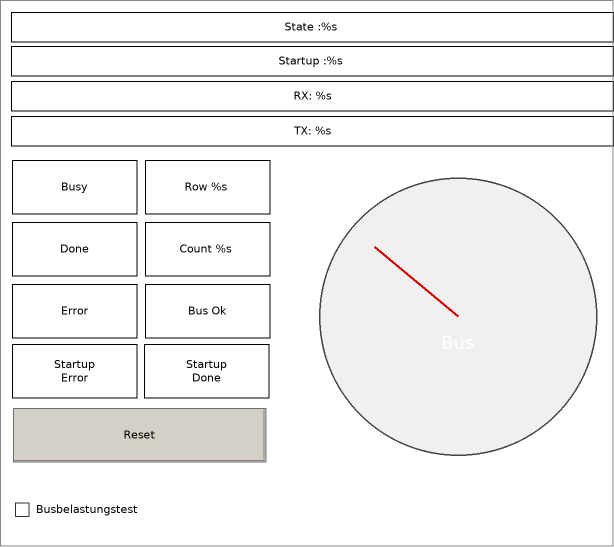
VISUALIZATION BusRS485Master_Frame  // 614x547
VAR_IN_OUT	
	(* für RS485 FiFo Master *)
	bBusBelastungstest		:BOOL;
	bReset					:BOOL;
	
	stFiFoMasterState		:ST_FiFoMaster_State;
	stRS48StartupState		:ST_RS485Startup_State;
END_VAR
    Meter360 (319,170 278x293), value: stFiFoMasterState.lrBusAuslastung, style: Meter-Meter360-Gray, scale format: %.1f, scale 0..350
    Rectangle (11,81 603x30), "RX: %s", text variable: stFiFoMasterState.sReceiveString
    Checkbox (13,472 254x75), "Busbelastungstest", variable: bBusBelastungstest
    Rectangle (11,116 603x30), "TX: %s", text variable: stFiFoMasterState.sSendString
    Rectangle (11,12 603x30), "State :%s", text variable: stFiFoMasterState.sState
    Rectangle (12,160 125x54), "Busy", colour toggle: stFiFoMasterState.bBusy
    Rectangle (12,222 125x54), "Done", colour toggle: stFiFoMasterState.bDone
    Rectangle (12,284 125x54), "Error", colour toggle: stFiFoMasterState.bError
    Rectangle (145,160 125x54), "Row %s", text variable: stFiFoMasterState.iFiFoRow
    Rectangle (145,222 125x54), "Count %s", text variable: stFiFoMasterState.iFiFoCount
    Button (13,408 253x54), "Reset"
        tap bReset
    Label (383,328 150x30), "Bus"
    Rectangle (11,46 603x30), "Startup :%s", text variable: stRS48StartupState.sStartupState
    Rectangle (145,284 125x54), "Bus Ok", colour toggle: stRS48StartupState.BusOk
    Rectangle (144,344 125x54), "Startup Done", colour toggle: stRS48StartupState.bStartupDone
    Rectangle (12,344 125x54), "Startup Error", colour toggle: stRS48StartupState.bStartupError
END_VISUALIZATION

// ---- VISUs/HausBus_RS485/BusTatster6F_Frame.TcVIS
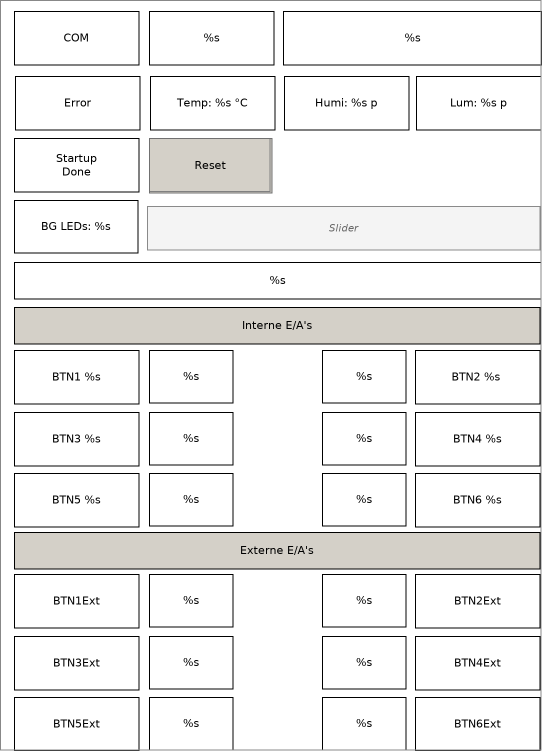
VISUALIZATION BusTatster6F_Frame  // 542x751
VAR_IN_OUT
	stBusTaster6F_Input		:ST_BusTaster6F_Input;
	stBusTaster6F_Output	:ST_BusTaster6F_Output;
	stBusTaster6F_Cnt		:ST_BusTaster6F_Cnt;
END_VAR
    Rectangle (14,11 125x54), "COM", colour toggle: stBusTaster6F_Output.bCOM
    Rectangle (14,350 125x54), "BTN1 %s", text variable: stBusTaster6F_Cnt.dwCntButtons[1], colour toggle: stBusTaster6F_Output.bButtons[1]
    Rectangle (149,11 125x54), "%s", text variable: stBusTaster6F_Input.diID
    Rectangle (283,11 259x54), "%s", text variable: stBusTaster6F_Input.sName
    Rectangle (415,350 125x54), "BTN2 %s", text variable: stBusTaster6F_Cnt.dwCntButtons[2], colour toggle: stBusTaster6F_Output.bButtons[2]
    Rectangle (14,412 125x54), "BTN3 %s", text variable: stBusTaster6F_Cnt.dwCntButtons[3], colour toggle: stBusTaster6F_Output.bButtons[3]
    Rectangle (415,412 125x54), "BTN4 %s", text variable: stBusTaster6F_Cnt.dwCntButtons[4], colour toggle: stBusTaster6F_Output.bButtons[4]
    Rectangle (14,473 125x54), "BTN5 %s", text variable: stBusTaster6F_Cnt.dwCntButtons[5], colour toggle: stBusTaster6F_Output.bButtons[5]
    Rectangle (415,473 125x54), "BTN6 %s", text variable: stBusTaster6F_Cnt.dwCntButtons[6], colour toggle: stBusTaster6F_Output.bButtons[6]
    Rectangle (149,350 84x53), "%s", text variable: stBusTaster6F_Input.iLED[1]
        OnMouseDown: write the text variable via VisuDialogs.Numpad, min 0, max 100
    Rectangle (322,350 84x53), "%s", text variable: stBusTaster6F_Input.iLED[2]
        OnMouseDown: write the text variable via VisuDialogs.Numpad, min 0, max 100
    Rectangle (149,412 84x53), "%s", text variable: stBusTaster6F_Input.iLED[3]
        OnMouseDown: write the text variable via VisuDialogs.Numpad, min 0, max 100
    Rectangle (322,412 84x53), "%s", text variable: stBusTaster6F_Input.iLED[4]
        OnMouseDown: write the text variable via VisuDialogs.Numpad, min 0, max 100
    Rectangle (149,473 84x53), "%s", text variable: stBusTaster6F_Input.iLED[5]
        OnMouseDown: write the text variable via VisuDialogs.Numpad, min 0, max 100
    Rectangle (322,473 84x53), "%s", text variable: stBusTaster6F_Input.iLED[6]
        OnMouseDown: write the text variable via VisuDialogs.Numpad, min 0, max 100
    Button (149,138 123x55), "Reset"
        tap stBusTaster6F_Input.bReset
    Rectangle (15,76 125x54), "Error", colour toggle: stBusTaster6F_Output.bError
    Rectangle (150,76 125x54), "Temp: %s °C", text variable: stBusTaster6F_Output.lrTemp
    Rectangle (284,76 125x54), "Humi: %s p", text variable: stBusTaster6F_Output.lrRhd
    Rectangle (416,76 125x54), "Lum: %s p", text variable: stBusTaster6F_Output.lrBrs
    Rectangle (14,262 527x37), "%s", text variable: stBusTaster6F_Output.sState
    Rectangle (14,138 125x54), "Startup Done", colour toggle: stBusTaster6F_Output.bStartupDone
    Rectangle (14,200 124x53), "BG LEDs: %s", text variable: stBusTaster6F_Input.iLEDBg
        OnMouseDown: write the text variable via VisuDialogs.Numpad, min 0, max 100
    Rectangle (14,574 125x54), "BTN1Ext", colour toggle: stBusTaster6F_Output.bButtonsExt[1]
    Rectangle (415,574 125x54), "BTN2Ext", colour toggle: stBusTaster6F_Output.bButtonsExt[2]
    Rectangle (14,636 125x54), "BTN3Ext", colour toggle: stBusTaster6F_Output.bButtonsExt[3]
    Rectangle (415,636 125x54), "BTN4Ext", colour toggle: stBusTaster6F_Output.bButtonsExt[4]
    Rectangle (14,697 125x54), "BTN5Ext", colour toggle: stBusTaster6F_Output.bButtonsExt[5]
    Rectangle (415,697 125x54), "BTN6Ext", colour toggle: stBusTaster6F_Output.bButtonsExt[6]
    Rectangle (149,574 84x53), "%s", text variable: stBusTaster6F_Input.iLEDExt[1]
        OnMouseDown: write the text variable via VisuDialogs.Numpad, min 0, max 100
    Rectangle (322,574 84x53), "%s", text variable: stBusTaster6F_Input.iLEDExt[2]
        OnMouseDown: write the text variable via VisuDialogs.Numpad, min 0, max 100
    Rectangle (149,636 84x53), "%s", text variable: stBusTaster6F_Input.iLEDExt[3]
        OnMouseDown: write the text variable via VisuDialogs.Numpad, min 0, max 100
    Rectangle (322,636 84x53), "%s", text variable: stBusTaster6F_Input.iLEDExt[4]
        OnMouseDown: write the text variable via VisuDialogs.Numpad, min 0, max 100
    Rectangle (149,697 84x53), "%s", text variable: stBusTaster6F_Input.iLEDExt[5]
        OnMouseDown: write the text variable via VisuDialogs.Numpad, min 0, max 100
    Rectangle (322,697 84x53), "%s", text variable: stBusTaster6F_Input.iLEDExt[6]
        OnMouseDown: write the text variable via VisuDialogs.Numpad, min 0, max 100
    Rectangle (14,532 526x37), "Externe E/A's"
    Rectangle (14,307 526x37), "Interne E/A's"
    Slider (147,206 393x44), variable: stBusTaster6F_Input.iLEDBg, scale 0..100
END_VISUALIZATION

// ---- VISUs/HausBus_RS485/RS485HB_ServiceVISU.TcVIS
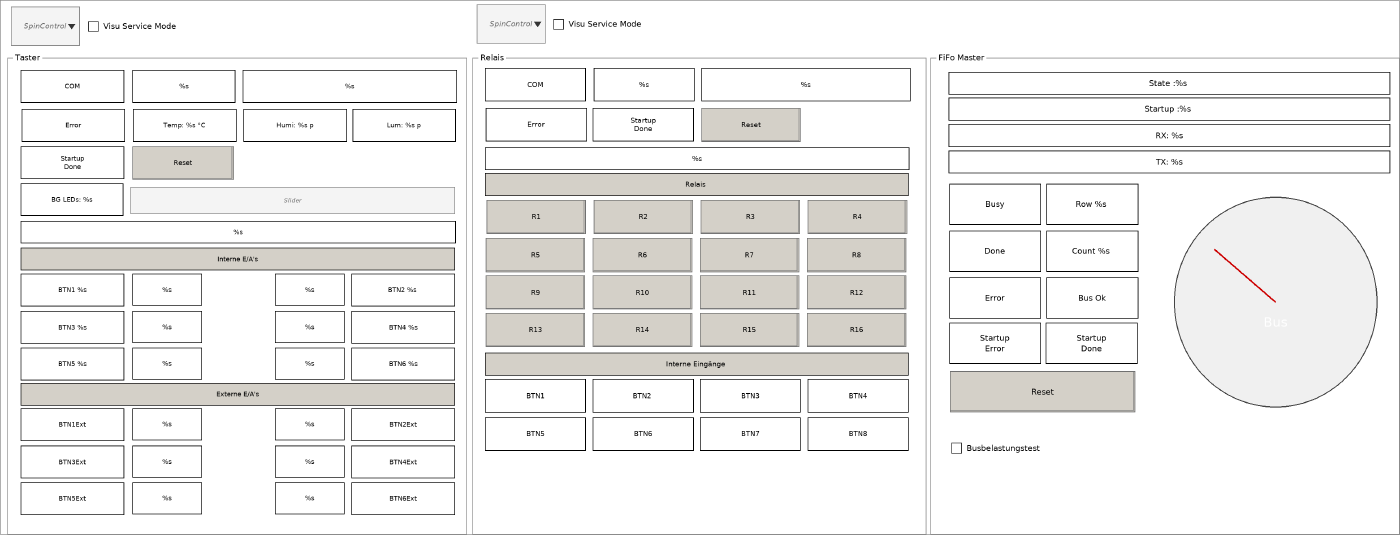
VISUALIZATION RS485HB_ServiceVISU  // 1938x741
    SpinControl (15,9 95x54), variable: GVL_ServiceVisu.iDeviceTasterVisu
        p651134158: cMaxBusTaster
    Checkbox (120,7 181x59), "Visu Service Mode", variable: GVL_ServiceVisu.bTasterServiceAktiv[GVL_ServiceVisu.iDeviceTasterVisu]
    SpinControl (660,6 95x54), variable: GVL_ServiceVisu.iDeviceRelaisVisu
        p576042468: cMaxBusTaster+1
        p651134158: cMaxBusRelais +cMaxBusTaster +1
    Checkbox (764,4 181x59), "Visu Service Mode", variable: GVL_ServiceVisu.bRelaisServiceAktiv[GVL_ServiceVisu.iDeviceRelaisVisu]
    GroupBox (654,72 628x669), "Relais"
        Frame (2,13 604x539)
            shows BusRelais16F_Frame(ST_BusRelais16F_Input := GVL_ServiceVisu.stRelaisService[GVL_ServiceVisu.iDeviceRelaisVisu], ST_BusRelais16F_Output := RS485_COM_PRG.fbRelais[GVL_ServiceVisu.iDeviceRelaisVisu].Q_stOutput, ST_BusRelais16F_Cnt := RS485_COM_PRG.fbRelais[GVL_ServiceVisu.iDeviceRelaisVisu].Q_stCnt)
    GroupBox (10,72 636x669), "Taster"
        Frame (3,16 619x625)
            shows BusTatster6F_Frame(stBusTaster6F_Input := GVL_ServiceVisu.stTasterService[GVL_ServiceVisu.iDeviceTasterVisu], stBusTaster6F_Output := RS485_COM_PRG.fbTaster[GVL_ServiceVisu.iDeviceTasterVisu].Q_stOutput, stBusTaster6F_Cnt := RS485_COM_PRG.fbTaster[GVL_ServiceVisu.iDeviceTasterVisu].Q_stCnt)
    GroupBox (1288,72 650x669), "FiFo Master"
        Frame (14,15 622x573)
            shows BusRS485Master_Frame(bBusBelastungstest := RS485_COM_PRG.fbRS485SendCmdFiFo.I_bBusBelastungstest, bReset := RS485_COM_PRG.fbRS485SendCmdFiFo.I_bReset, stFiFoMasterState := RS485_COM_PRG.fbRS485SendCmdFiFo.Q_stStates, stRS48StartupState := RS485_COM_PRG.fbRS485Startup.Q_stStates)
            shows BusRS485Master_Frame()
END_VISUALIZATION
